TYPE HMIButtonNumericalInputInterface :
STRUCT
	IsEnabled	:	BOOL;
	IsPressed	:	BOOL;
	InPosition	:	BOOL;
	IsVisibleButton	:	BOOL;
	CaptionButton	:	STRING;
	PathImageButton	:	STRING;
END_STRUCT
END_TYPE

(* stored: Version 1.1.0.1
   DUT HMIButtonNumericalInputInterface: Id {9cc8cd21-676b-4a52-9373-99f7a05031db} *)
